TYPE ST_SafetyIn :
STRUCT
    stMCCStatusIn: ST_MCCStatusIn;
    stMCC_CustomStatusIn: ST_MCC_CustomStatusIn;
    astSafetyFunctionIn: ARRAY[1..GVL_SafetyIO.cNBR_OF_SF] OF ST_SafetyFunctionIn;
    stLEDState: ST_LEDState;

    astTechnosoftIn: ARRAY[1..GVL_SafetyIO.cNBR_OF_TECHNOSOFT] OF ST_TechnosoftIn;
    astTechnosoftMotionError: ARRAY[1..GVL_SafetyIO.cNBR_OF_TECHNOSOFT] OF ST_TechnosoftMotionError;
END_STRUCT
END_TYPE

(* stored: Version 1.1.0.1
   DUT ST_SafetyIn: Id {fc6082d6-fb28-0397-2e5b-2e7f309b5b60} *)
